(*udt (user defined type) of Beckhoff EP6224-0002 - 4 Point IP67 Rated IO-Link Box:
	Version 20190506
		- initial creation, j.vandongen


*)


TYPE udt_EP6224_CMD :
STRUCT
	Port1_Q: BOOL;
	Port2_Q: BOOL;
	Port3_Q: BOOL;
	Port4_Q: BOOL;

END_STRUCT
END_TYPE

(* stored: Version 1.1.0.1, ProductVersion 3.1.4024.9
   DUT udt_EP6224_CMD: Id {93c22185-468c-4829-af42-e83dd0fc70b0} *)
